{attribute 'qualified_only'}
{attribute 'strict'}
TYPE Main_STM :
(
  Init,
  Run,
  FillingArrays,
  SearchIndex,
  Idle,
  Error
);
END_TYPE

(* stored: Version 1.1.0.1, ProductVersion 3.1.4024.12
   DUT Main_STM: Id {b2e29890-c613-43ea-860c-b9efeb22fffc} *)
